Fanuc KAREL source: kd00056.KL

-- PROVISIONAL review KL for V940-1; original PC SHA256 d5aec94cb6d650456eb744e25d159b5f479bf486a91fd22d0a4730e27c9b7db2
-- Incomplete behavior may be omitted. Consult companion uncertainty JSON. Do not deploy.
PROGRAM KD00056
%NOLOCKGROUP
VAR
  I : INTEGER
  J : INTEGER
  B : BOOLEAN
  R : REAL
  S : STRING[80]
-- UNRESOLVED_DECL P type=000101
BEGIN
  -- V9_ZERO_TABLE_METADATA_HINT layout=0001; no indexed target words; source/name/runtime held
  -- UNRESOLVED_PC offsets 5-37; opcodes 01,22,1C,06,82,03,9D,9C,9D,12,9D,1B,9D,13,04,0B
  -- UNRESOLVED_PC offsets 42-46; opcodes 7F
END KD00056
